// TIA Portal V17 export
// export: Created 2025-03-10T13:12:21.3449745Z, ExportSetting WithDefaults, DisplayName Totally Integrated Automation Portal, DisplayVersion V17 Update 8, DisplayName TIA Portal Openness, DisplayVersion V17 Update 8, DisplayName TIA Portal Version Control Interface, DisplayVersion V17, DisplayName SINAMICS Startdrive Advanced, DisplayVersion V17 SP2, DisplayName SINAMICS Startdrive G110M, G120, G120C, G120D, G120P, G115D, DisplayVersion V17 SP2, DisplayName SINAMICS Startdrive G130, G150, S120, S150, SINAMICS MV, S210, DisplayVersion V17 SP2, DisplayName STEP 7 Professional, DisplayVersion V17 Update 8, DisplayName SINUMERIK ONE STEP 7 Toolbox, DisplayVersion V17 Update 12, DisplayName SINUMERIK 840D sl STEP 7 Toolbox, DisplayVersion V17 Update 12, DisplayName STEP 7 Safety, DisplayVersion V17 Update 6, DisplayName WinCC Advanced, DisplayVersion V17 Update 8
TYPE "POWDER FEEDER HMI OFFSETS ALARMS WARNINGS"
// stored: IsFailsafeCompliant false
   STRUCT
      CarrierGasNominalLine1_Max_Alarm : Real;
      CarrierGasNominalLine2_Max_Alarm : Real;
      DiskSpeedNominalLine1_Max_Alarm : Real;
      DiskSpeedNominalLine2_Max_Alarm : Real;
      StirrerSpeedNominalLine1_Max_Alarm : Real;
      StirrerSpeedNominalLine2_Max_Alarm : Real;
      HopperTempNominalLine1_Max_Alarm : Real;
      HopperTempNominalLine2_Max_Alarm : Real;
      CarrierGasNominalLine1_Min_Alarm : Real;
      CarrierGasNominalLine2_Min_Alarm : Real;
      DiskSpeedNominalLine1_Min_Alarm : Real;
      DiskSpeedNominalLine2_Min_Alarm : Real;
      StirrerSpeedNominalLine1_Min_Alarm : Real;
      StirrerSpeedNominalLine2_Min_Alarm : Real;
      CarrierGasNominalLine1_Max_Warning : Real;
      CarrierGasNominalLine2_Max_Warning : Real;
      DiskSpeedNominalLine1_Max_Warning : Real;
      DiskSpeedNominalLine2_Max_Warning : Real;
      StirrerSpeedNominalLine1_Max_Warning : Real;
      StirrerSpeedNominalLine2_Max_Warning : Real;
      CarrierGasNominalLine1_Min_Warning : Real;
      CarrierGasNominalLine2_Min_Warning : Real;
      DiskSpeedNominalLine1_Min_Warning : Real;
      DiskSpeedNominalLine2_Min_Warning : Real;
      StirrerSpeedNominalLine1_Min_Warning : Real;
      StirrerSpeedNominalLine2_Min_Warning : Real;
      Spare26 : Real;
      Spare27 : Real;
      Spare28 : Real;
      Spare29 : Real;
      Spare30 : Real;
   END_STRUCT;
END_TYPE
